TYPE ST_Parameters :
STRUCT
	fCyclicTime 					: LREAL := 0.001; // [s]
	fMaxWinchVelocityLimit 			: LREAL := 0.025; // [m/s]
	bWinchDeadBandCompOn 			: BOOL := FALSE;
	bDisplacementDeadBandCompOn 	: BOOL := FALSE;
	stWinchValveDeadBand 			: ST_ValveDeadBand := (fPosMax := 32767.0, fPosMin := 16383.0, fNegMin := 16383.0, fNegMax := 0);
	stDisplacementValveDeadBand 	: ST_ValveDeadBand := (fPosMax := 32767.0, fPosMin := 16383.0, fNegMin := 16383.0, fNegMax := 0);
	stPressureSensorScaling400bar 	: ST_AnalogInputScaling := (fMaxInputValue := 32767.0, fMinInputValue := 0.0, fMaxOutputValue := 400.0, fMinOutputValue := 0.0);
	stPressureSensorScaling40bar 	: ST_AnalogInputScaling := (fMaxInputValue := 32767.0, fMinInputValue := 0.0, fMaxOutputValue := 40.0, fMinOutputValue := 0.0);
	stJoystickInputScalingX 		: ST_JoystickInputScaling := (fMaxInputValue := 14790.0, fMinInputValue := 1797.0, fNeutralInputValue := 8400, fNeutralDeadband := 50.0, fMaxOutputValue := 1.0, fMinOutputValue := -1.0, fNeutralOutputValue := 0.0);
	stJoystickInputScalingY 		: ST_JoystickInputScaling := (fMaxInputValue := 14770.0, fMinInputValue := 1829.0, fNeutralInputValue := 8340, fNeutralDeadband := 50.0, fMaxOutputValue := 1.0, fMinOutputValue := -1.0, fNeutralOutputValue := 0.0);
	stJoystickInputScalingZ 		: ST_JoystickInputScaling := (fMaxInputValue := 14830.0, fMinInputValue := 1804.0, fNeutralInputValue := 8380, fNeutralDeadband := 50.0, fMaxOutputValue := 1.0, fMinOutputValue := -1.0, fNeutralOutputValue := 0.0);
	fWinchEncoderOffset 			: LREAL := -5886686.1725795381; // Encoder value at zero (Cylinder out / second layaer)
	stYokeInputScaling 				: ST_YokeInputScaling := (fMaxInputValue := 25000.0, fMinInputValue := 6150.0, fNeutralInputValue := 15470, fNeutralDeadband := 0.0, fMaxOutputValue := 1.0, fMinOutputValue := -1.0, fNeutralOutputValue := 0.0);
	fDisplacementControlPgain 		: LREAL := 2.0; /// HER Er Daines Gain ///
	fWinchDrumRadius 				: LREAL := 0.075;
	fWinchEndStopPos 				: LREAL := 2.16;
	fWinchEndStopNeg 				: LREAL := 1.0;
	fPayloadMass 					: LREAL := 78.0; 
END_STRUCT
END_TYPE

(* stored: Version 1.1.0.1, ProductVersion 3.1.4024.12
   DUT ST_Parameters: Id {a43a257d-4d38-4d6a-971b-afd17eab7788} *)
